// TwinCAT 3 PLC project plc1
// ProgramVersion: 3.1.4023.0
// libraries:
//   Tc2_Standard, * (Beckhoff Automation GmbH)
//   Tc2_System, * (Beckhoff Automation GmbH)
//   Tc2_Utilities, * (Beckhoff Automation GmbH)
//   Tc3_EventLogger, * (Beckhoff Automation GmbH)
//   Tc3_Module, * (Beckhoff Automation GmbH)
//   Tc3_Vision, * (Beckhoff Automation GmbH)
// project tree:
//   / GlobalTextList.TcGTLO, PlcTask.TcTTO, Visualization Manager.TcVMO (not stored)
//   GVLs/ GVL_VideoPlaybackConfig.TcGVL
//   POUs/ FB_CreateVidOnAlarm.TcPOU, MAIN.TcPOU, ScopeRecordTestCode.TcPOU
// real-time tasks:
//   TASK PlcTask: cycle T#10ms, priority 20, ADS port 350
//   TASK VnTask ImgAcq (Camera1): cycle T#1ms, priority 5, ADS port 351
//   TASK VnTask ADS (Camera1): cycle T#10ms, priority 6, ADS port 352
//   TASK Task 6: cycle default, priority 1
//   TASK Task 7: cycle default, priority 2
//   TASK VISU_TASK: cycle T#200000us, priority 30, ADS port 353

CONFIGURATION plc1
    RESOURCE PLC ON TwinCAT3
        TASK PlcTask(INTERVAL := T#10ms, PRIORITY := 20);
        PROGRAM MAIN WITH PlcTask : MAIN;
    END_RESOURCE
END_CONFIGURATION

// ---- GVLs/GVL_VideoPlaybackConfig.TcGVL
{attribute 'qualified_only'}
VAR_GLOBAL
END_VAR

// ---- POUs/MAIN.TcPOU
PROGRAM MAIN
VAR
	hr					:	HRESULT;	// ADS return code in hex 16#....70C -> didn't get new image, 000 means all good, success
	fbCamera			:	FB_VN_SimpleCameraControl;
	eState				:	ETcVnCameraState;
	
	// Images
	ipImageIn			:	ITcVnImage;
	ipImageInDisp		:	ITcVnDisplayableImage;
	ipImageWork			:	ITcVnImage;
	ipImageResultDisp	:	ITcVnDisplayableImage;
END_VAR

//call test PRG
ScopeRecordTestCode();


//code to control the camera, puts in acquisition mode and brings in images. 
eState:=fbCamera.GetState();
	
CASE eState OF

	TCVN_CS_INITIAL,
	TCVN_CS_OPENING,
	TCVN_CS_OPENED,
	TCVN_CS_STARTACQUISITION:
		hr:= fbCamera.StartAcquisition();
	
	TCVN_CS_ACQUIRING:
		hr:= fbCamera.GetCurrentImage(ipImageIn);
		IF SUCCEEDED(hr) THEN
			// display
			hr:= F_VN_CopyIntoDisplayableImage(ipImageIn, ipImageInDisp, hr);
				hr:= F_VN_ConvertColorSpace(ipImageIn, ipImageWork, TCVN_CST_Bayer_RG_TO_RGB, hr);
				hr:= F_VN_CopyIntoDisplayableImage(ipImageWork, ipImageResultDisp, hr);
		END_IF
END_CASE

ACTION aNotes:
(*

HRESULT
All TwinCAT Vision functions return an HRESULT after their execution. Its value indicates whether the
execution was successful or not.

16#NXXXXCCC ==> Value of N indicates success or failure

SUCCESS codes
A successful execution is indicated by a POSITVE code. In hexadecimal notation the first digit (N) is between 0 and 7.
Frequent SUCCESS codes are:

Code 		Name 				Description
CCC = 000 	S_OK 				Function was executed successfully
CCC = 001 	S_FALSE 			Function was executed successfully but did not reach a complete result. 
								(Occurs, for example, with the Code Reading functions if no code was found in the image.)
CCC = 203 	S_PENDING 			Asynchronous method was started but there is no result yet 
								(Occurs at the first call of fbCameraControl.StartAcquisition(), for example; at the second call S_OK is returned, for example)
CCC = 256 	S_WATCHDOGTIMEOUT	Function was aborted by the watchdog.

ERROR codes
A failed execution is indicated by a NEGATIVE code, or in hexadecimal notation the first digit (N) is >= 8. The
final digits of the code correspond to the ADS Return Code.
NOTE If an error code is returned, it means that all returns of the function are invalid. and must therefore not be used.

Common ERROR codes with the TwinCAT Vision API elements are:
Code 	 	Name 				Description
CCC = 70A  	NOMEMORY 			Insufficient memory
CCC = 70B  	INVALIDPARM 		Invalid parameter values
CCC = 70C  	NOTFOUND 			Not found (file, image, ...)
CCC = 70E  	INCOMPATIBLE 		Objects do not match
CCC = 712  	INVALIDSTATE 		The method of an FB was called in an impermissible state.
CCC = 719  	TIMEOUT 			timeout
CCC = 71A  	NOINTERFACE 		Interface query failed
CCC = 71B  	INVALIDINTERFACE 	Wrong interface requested.
CCC = 71D  	INVALIDOBJID 		Object ID is invalid.
CCC = 734  	OUTOFRANGE 			Outside the valid range.

*)
END_ACTION

END_PROGRAM

// ---- POUs/ScopeRecordTestCode.TcPOU
PROGRAM ScopeRecordTestCode
VAR
	//Test Bits
	SomethingBadHappendOnMachine 	: BOOL;
	
	//Alarm init and handeling
	fbAlarm 		: FB_TcAlarm;
	bIsInitalized 	: BOOL;
	bRaiseAlarm		: BOOL;
	hr				: HRESULT;
	hrLastError		: HRESULT;
	//string used to determine if this particular alarm should generate a video or not. 
	JSONString		: STRING := '{"CreateVideo": 1}';
	
	VideoDestinationPath	: STRING(255) := 'C:\Temp\Scope Project_Img_test\';
	ScopeImageExportPath	: STRING(255) := 'C:\Temp\Scope Project_Img_test\ipImageResultDisp\';
	
	EventTimestamp: TimeStruct;
	bConfirmAlarm: BOOL;
	bClearAlarm: BOOL;
	
	sTEMP			: STRING;
	sFileName		: STRING;
	RecordCreated	: BOOL;
	sDump			: STRING;	
	fbCreateVideoOnAlarm		: FB_CreateVidOnAlarm;
	
	AlarmCount: INT;
END_VAR

IF NOT bIsInitalized THEN
	bIsInitalized := TRUE;
	hr := fbAlarm.CreateEx(TC_EVENTS.VideoAlarmDemoEventClass.MachineError, TRUE, 0);
	IF FAILED(hr) THEN
		hrLastError := hr;
	END_IF
END_IF

//cyclic call to FB watch for events
fbCreateVideoOnAlarm(
	ImageExportPath:= ScopeImageExportPath,  //this needs to match the image export path in scope trigger
	VideoDestinationPath:= VideoDestinationPath, //this should match the virtual directory set in TC HMI to be able to find the video file.
	JSONAttribute:= JSONString, 
	//sFileName:= sFileName, 
	bBusy=> , 
	bError=> , 
	nErrID=> );

//Something did not go as planned in the machine sequence, raise an alarm, and associate the video JSON attribute to the riased alarm
	//SomethingBadHappendOnMachine:=FALSE;
IF SomethingBadHappendOnMachine THEN
	hr:= fbAlarm.SetJsonAttribute(JSONSTRING);
	hr:= fbAlarm.Raise(0);
	IF FAILED(hr) THEN
		hrLastError := hr;
	END_IF
END_IF


IF bConfirmAlarm THEN
	fbAlarm.Confirm(0);
	fbAlarm.Clear(0, FALSE);
	bConfirmAlarm := FALSE;
END_IF

END_PROGRAM

// ---- POUs/FB_CreateVidOnAlarm.TcPOU
FUNCTION_BLOCK FB_CreateVidOnAlarm EXTENDS FB_ListenerBase2
VAR_INPUT
	ImageExportPath			: T_MaxString;
	VideoDestinationPath	: T_MaxString;
	JSONAttribute			: T_MaxString;	

END_VAR
VAR_OUTPUT
	bBusy 	: BOOL;
	bError 	: BOOL;
	nErrID 	: UDINT;
END_VAR
VAR
	//Settings creation of the Video
	BatchFileFullPath: STRING := 'C:\TwinCAT\3.1\Boot\Images2Video.bat'; //Full Path to Batch file
	DelayTimebeforeCallingBatch : TIME := T#15S; //Delay time after alarm trigger, this value should match the 'post' trigger time in scope image export trigger
	
	//text retrieval of message
	fbRequestEventText : FB_RequestEventText;
	{attribute 'TcEncoding':='UTF-8'}
	sLastMessageText : STRING;
	bReqText : BOOL;
	
	
	//Internal Vars
	CallBatchFile 		: NT_StartProcess;
	BatchFileDelay		: TON;
	Command 			: STRING(1000);	
	TriggerVideoCreate	: BOOL;	
	JSONFilter			: FB_TcEventFilter;
	hr					: HRESULT;
	sFileName			: T_MaxString;
	EventTimestamp		: TimeStruct;
	sDump				: STRING;
	_fbEvent 			: FB_TcEvent;
	NumAlarmsRaised		: INT := 0;
	nCntAlarmsRaised	: INT;
	Step				:INT;
	sJsonAttribute 		: STRING (10000);	
	bSubscribe			: BOOL :=TRUE;
	bSubscribed			: BOOL;
	bUnSubscribe		: BOOL;
END_VAR

Execute();


IF bSubscribe THEN 
	bSubscribe := FALSE;
	JSONFilter.Clear().JsonAttribute.Value.EqualTo(JSONAttribute); //define all events (messages and alarms) from this eventclass   
	hr := Subscribe2(JSONFilter); //subscribe to retrieve defined events
	IF SUCCEEDED(hr) THEN	
		bSubscribed := TRUE;
	END_IF
END_IF 

IF bUnSubscribe THEN 
	bUnSubscribe := FALSE;
	hr := Unsubscribe();
	IF SUCCEEDED(hr) THEN	
		bSubscribed := FALSE;
	END_IF
END_IF 

(*
IF nAlarms <> NumAlarmsRaised THEN
	NumAlarmsRaised := NumAlarmsRaised + 1;
	TriggerVideoCreate := TRUE;
END_IF
*)

CASE Step OF
	0: 
		IF TriggerVideoCreate THEN
			EventTimestamp := FILETIME64_TO_SYSTEMTIME(_fbevent.nTimestamp);
			//CreateVideo(ImageExportPath := ScopeImageExportPath, VideoDestinationPath := VideoDestinationPath, JSONAttribute := JSONString);
		
		//Get timestamp, convert it to a format that can be used for a file name, and build up the filename for the video
			sFileName := SYSTEMTIME_TO_STRING(EventTimestamp);
			FindAndReplaceChar(ADR(sFileName),':','-',ADR(sFileName),SIZEOF(sFileName));
			sFileName := sFileName;
			FindAndSplitChar(sSeparatorChar:='.',pSrcString:= ADR(sFileName),pLeftString :=ADR(sFileName),
			nLeftSize:= SIZEOF(FileName), pRightString := ADR(sDump), nRightSize := SIZEOF(sDump),bSearchFromRight := FALSE);
		
			//Create Commandline agrument to call batch file will passed in args
			Command :='';
			Command := CONCAT(Command, ' "');
			Command := CONCAT(Command, sFileName);
			Command := CONCAT(Command, '" "');
			Command := CONCAT(Command, VideoDestinationPath);
			Command := CONCAT(Command, '" "');
			Command := CONCAT(Command, ImageExportPath);
			Command := CONCAT(Command, '"'); 
			
			bBusy := TRUE;
			Step:= Step+10;
		END_IF 

	10:
		//Call NT_StartProcess to make sure it's called with a False "Start"
			CallBatchFile(	PATHSTR:= BatchFileFullPath, 
						COMNDLINE := Command,
						START := FALSE);
		
		Step:= Step+10;
		
	20:
		IF BatchFileDelay.Q THEN
			CallBatchFile(	PATHSTR:= BatchFileFullPath, 
						COMNDLINE := Command,
						START := TRUE);
			BatchFileDelay(IN := FALSE);
			CallBatchFile(START := FALSE);
			bBusy := FALSE;
			nErrID := 0;
			TriggerVideoCreate := FALSE;
			
			Step:=0;
		END_IF
	
END_CASE

//Delay time after alarm trigger, this value should match the 'post' trigger time in scope image export trigger
		BatchFileDelay(IN:= TriggerVideoCreate,PT := DelayTimebeforeCallingBatch);

METHOD Execute : HRESULT
VAR_INPUT
END_VAR
Execute := SUPER^.Execute(); //retrieve events

//retrieve the text of a message
IF 	bReqText AND fbRequestEventText.bError THEN 
	sLastMessageText := 'Error';
	bReqText := FALSE; 
ELSIF bReqText AND NOT  fbRequestEventText.bBusy THEN
	fbRequestEventText.GetString(sLastMessageText, SIZEOF(sLastMessageText));
	bReqText := FALSE;
END_IF
END_METHOD

METHOD OnAlarmRaised : HRESULT
VAR_INPUT
	fbEvent	: REFERENCE TO FB_TcEvent;
END_VAR


TriggerVideoCreate := TRUE;
_fbEvent:=fbevent;

hr := fbEvent.GetJsonAttribute(sJsonAttribute, SIZEOF(sJsonAttribute));
nCntAlarmsRaised := nCntAlarmsRaised + 1;

OnAlarmRaised := S_OK; // in order to receive more callbacks (Set <> S_OK in order to cancel the callbacks for this program cycle.)
END_METHOD

END_FUNCTION_BLOCK
